# EPICS substitutions: evrSupport/Db/ioc/IOC-LI21-BL01bsa.substitutions
# BSA records
#
# One per IOC:
#
file bsaEdefShadow.db {
  pattern { DEVICE       , SYSI }
          { IOC:LI21:BL01, SYS0 }
}

# One per device:
# Please check the HOPR,LOPR,PREC,ADEL,MDEL values provided in bsaBPMSEdef.db!
file bsaBPMSEdef.db {
#      Device        ,loc'n , IOC unit, timing system
  pattern {DEVICE    , LOC  ,  UN  , SYS  }
	  { BLEN:LI21:265, LI21 , BL01 , SYS0 }
	  { BLEN:LI21:280, LI21 , BL01 , SYS0 }
}
